TYPE DUT_UpdateBroachingProfileSettings :
STRUCT
	IdBroachingProfileSettings	: DINT;
	DataBroachingProfile		: STRING(DB.MAX_STRING_SIZE);
END_STRUCT
END_TYPE

(* stored: Version 1.1.0.1, ProductVersion 3.1.4024.15
   DUT DUT_UpdateBroachingProfileSettings: Id {da0974af-f421-4829-b9f7-eba5ff8dbd57} *)
